FUNCTION_BLOCK AX_ATM_FB_TON_REST (* AX_ATM_FB_TON, zusaetzlich mit REST (verbleibende Zeit PT-ET) als AR-Ausgang *)
  (* Standard: 61131-3; Classification: standard timer function block; Description: Copyright (c) 2026 HR Agrartechnik GmbH This program and the accompanying materials are made available under the terms of the Eclipse Public License 2.0 which is available at https://www.eclipse.org/legal/epl-2.0/ SPDX-License-Identifier: EPL-2.0 Kapselt die in mehreren Anwendungen wiederkehrende Kette AX_ATM_FB_TON -> ATM_SUB(PT,ET) -> ATM_IN_S_TO_ALR -> ALR_TO_AR in einem Baustein. REST ist die verbleibende Zeit in Sekunden (PT-ET), ohne Sentinel-Konvention (kein -1 bei inaktiv) - ein Aufrufer, der z.B. -1=inaktiv braucht, gated REST selbst mit einem AR_AX_SEL_AR davor/danach. REST aktualisiert sich mit derselben Aufloesung wie ET (E_D_FF_ANY, nur bei tatsaechlicher Wertaenderung von ET oder PT). *)
  (* Version 1.0, 2026-08-26, Franz Höpfinger, HR Agrartechnik GmbH, initial API and implementation *)
  PACKAGE adapter::iec61131::timers;
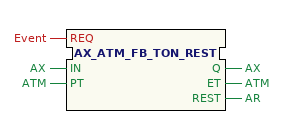
  EVENT_INPUT
    REQ; (* wie AX_ATM_FB_TON.REQ - gleichwertig zu IN.E1/PT.E1 *)
  END_EVENT
  SOCKETS
    IN : adapter::types::unidirectional::AX; (* Input *)
    PT : adapter::types::unidirectional::ATM; (* Process time *)
  END_SOCKETS
  PLUGS
    Q : adapter::types::unidirectional::AX; (* Output *)
    ET : adapter::types::unidirectional::ATM; (* Elapsed time *)
    REST : adapter::types::unidirectional::AR; (* Verbleibende Zeit PT-ET, Sekunden, kein Sentinel *)
  END_PLUGS
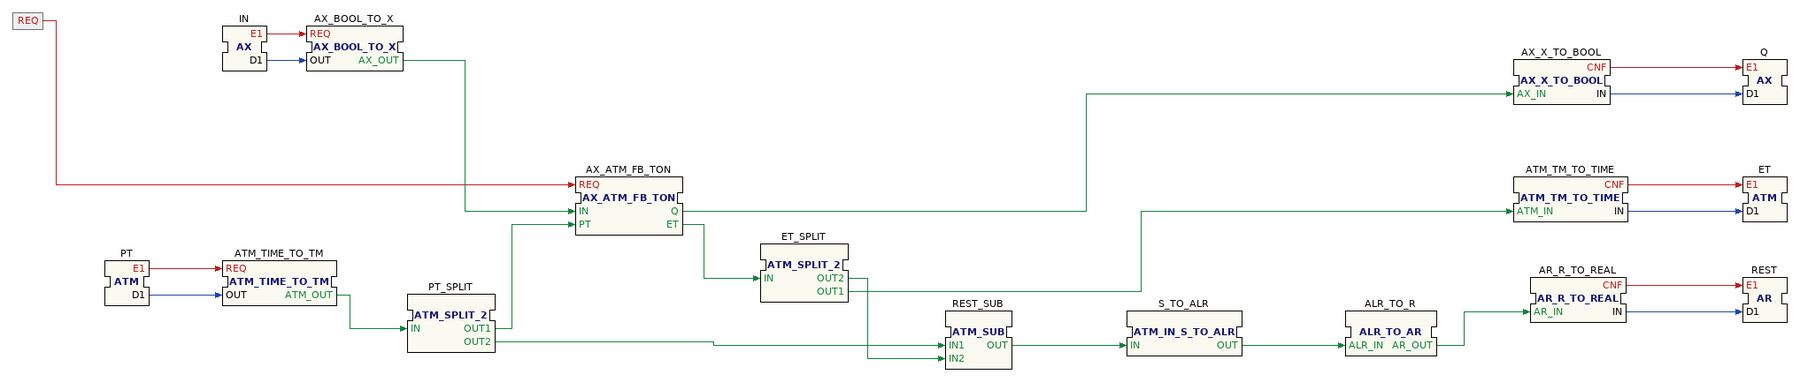
  FBS
    AX_ATM_FB_TON : adapter::iec61131::timers::AX_ATM_FB_TON;
    PT_SPLIT : adapter::events::unidirectional::ATM_SPLIT_2;
    ET_SPLIT : adapter::events::unidirectional::ATM_SPLIT_2;
    REST_SUB : adapter::iec61131::arithmetic::ATM_SUB;
    S_TO_ALR : adapter::conversion::unidirectional::ATM_IN_S_TO_ALR;
    ALR_TO_R : adapter::conversion::unidirectional::ALR_TO_AR;
    AR_R_TO_REAL : adapter::conversion::unidirectional::AR_R_TO_REAL;
    AX_X_TO_BOOL : adapter::conversion::unidirectional::AX_X_TO_BOOL;
    ATM_TM_TO_TIME : adapter::conversion::unidirectional::ATM_TM_TO_TIME;
    AX_BOOL_TO_X : adapter::conversion::unidirectional::AX_BOOL_TO_X;
    ATM_TIME_TO_TM : adapter::conversion::unidirectional::ATM_TIME_TO_TM;
  END_FBS
  EVENT_CONNECTIONS
    REQ TO AX_ATM_FB_TON.REQ;
    AR_R_TO_REAL.CNF TO REST.E1;
    AX_X_TO_BOOL.CNF TO Q.E1;
    ATM_TM_TO_TIME.CNF TO ET.E1;
    IN.E1 TO AX_BOOL_TO_X.REQ;
    PT.E1 TO ATM_TIME_TO_TM.REQ;
  END_CONNECTIONS
  DATA_CONNECTIONS
    AR_R_TO_REAL.IN TO REST.D1;
    AX_X_TO_BOOL.IN TO Q.D1;
    ATM_TM_TO_TIME.IN TO ET.D1;
    IN.D1 TO AX_BOOL_TO_X.OUT;
    PT.D1 TO ATM_TIME_TO_TM.OUT;
  END_CONNECTIONS
  ADAPTER_CONNECTIONS
    PT_SPLIT.OUT1 TO AX_ATM_FB_TON.PT;
    PT_SPLIT.OUT2 TO REST_SUB.IN1;
    AX_ATM_FB_TON.ET TO ET_SPLIT.IN;
    ET_SPLIT.OUT2 TO REST_SUB.IN2;
    REST_SUB.OUT TO S_TO_ALR.IN;
    S_TO_ALR.OUT TO ALR_TO_R.ALR_IN;
    ALR_TO_R.AR_OUT TO AR_R_TO_REAL.AR_IN;
    AX_ATM_FB_TON.Q TO AX_X_TO_BOOL.AX_IN;
    ET_SPLIT.OUT1 TO ATM_TM_TO_TIME.ATM_IN;
    AX_BOOL_TO_X.AX_OUT TO AX_ATM_FB_TON.IN;
    ATM_TIME_TO_TM.ATM_OUT TO PT_SPLIT.IN;
  END_CONNECTIONS
END_FUNCTION_BLOCK
